FUNCTION EncoderConvert : LREAL
VAR_INPUT
	iEncoderValue : UDINT;
END_VAR
VAR
	//CONSTANTS
	ENCODER_OFFSET : UDINT := 1305092900;
	ENCODER_CONVERSION : UDINT := 1637500000*180;
END_VAR

//convert raw value to Degrees
EncoderConvert := DINT_TO_LREAL(UDINT_TO_DINT(iEncoderValue) - 1305092900) / 163750000.0 * 180.0 / PI;

END_FUNCTION

(* stored: Version 1.1.0.1
   POU EncoderConvert: Id {257166ef-8fe7-4f81-8d05-dfb44ef5b943}, SpecialFunc None *)
